PROGRAM P3_03_ProcessData
VAR
	stDBParam 					:ST_ProcessData;	

	fbDBWrite					:FB_PLCDBWriteEvt(sNetId:=CONST.AMS_NETID, tTimeout:=DEFAULT_ADS_TIMEOUT);
	tableColumns				:ARRAY [0..8] OF STRING(50) := ['Batch', 'DateTime', 'Value1', 'Value2', 'Value3', 'Value4', 'Value5', 'Value6', 'Value7'];
	arrParam					:ARRAY [0..8] OF ST_ExpParameter := [(sParaName := 'Batch', nParaSize := 101, eParaType := E_EXPPARAMETERTYPE.STRING_),
															 (sParaName := 'DateTime', nParaSize := 4, eParaType := E_EXPPARAMETERTYPE.DateTime), 
															 (sParaName := 'Value1', nParaSize := 101, eParaType := E_EXPPARAMETERTYPE.STRING_), 
															 (sParaName := 'Value2', nParaSize := 101, eParaType := E_EXPPARAMETERTYPE.STRING_), 
															 (sParaName := 'Value3', nParaSize := 101, eParaType := E_EXPPARAMETERTYPE.STRING_),
															 (sParaName := 'Value4', nParaSize := 101, eParaType := E_EXPPARAMETERTYPE.STRING_),
															 (sParaName := 'Value5', nParaSize := 101, eParaType := E_EXPPARAMETERTYPE.STRING_),
															 (sParaName := 'Value6', nParaSize := 101, eParaType := E_EXPPARAMETERTYPE.STRING_),
															 (sParaName := 'Value7', nParaSize := 101, eParaType := E_EXPPARAMETERTYPE.STRING_)];
		
	fbDeleteTable    			:FB_PLCDBCmdEvt(sNetID:=CONST.AMS_NETID, tTimeout:=DEFAULT_ADS_TIMEOUT);	
	sDelete						:STRING;	
	bDelete						:BOOL;
										 
	bWrite						:BOOL;	
	
	sChopper1Speed				:STRING;
	sChopper2Speed				:STRING;
END_VAR
VAR // added by the converter: edge detectors and wires of the graphical bodies
    _rt1, _rt2 : R_TRIG;
END_VAR

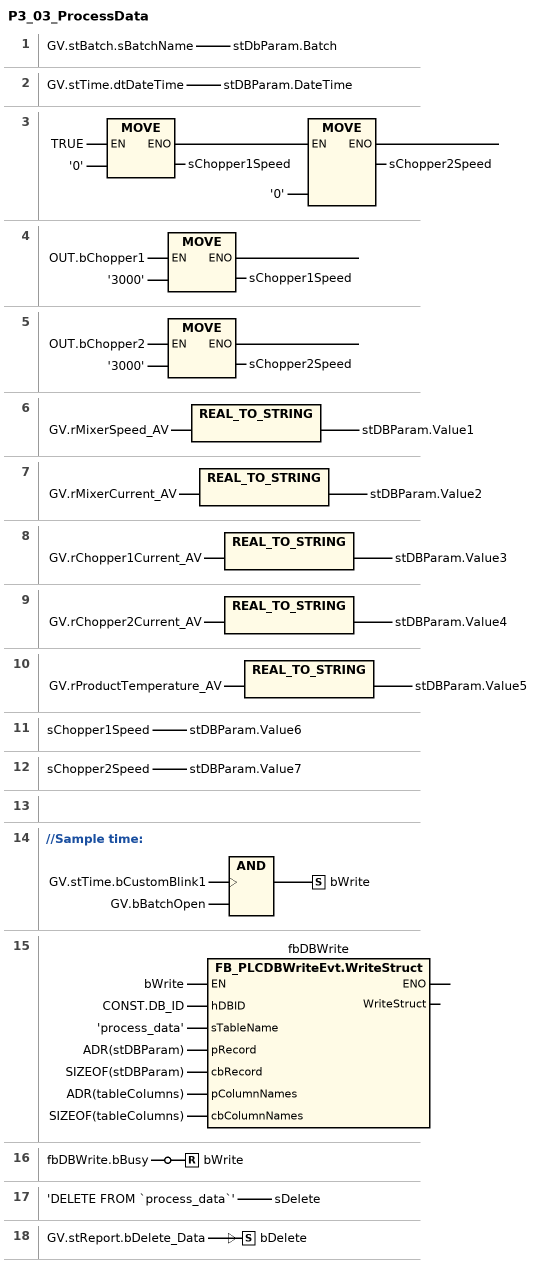
// NETWORK 1
stDbParam.Batch := GV.stBatch.sBatchName;

// NETWORK 2
stDBParam.DateTime := GV.stTime.dtDateTime;

// NETWORK 3
sChopper1Speed := '0';
sChopper2Speed := '0';

// NETWORK 4
IF OUT.bChopper1 THEN sChopper1Speed := '3000'; END_IF

// NETWORK 5
IF OUT.bChopper2 THEN sChopper2Speed := '3000'; END_IF

// NETWORK 6
stDBParam.Value1 := REAL_TO_STRING(GV.rMixerSpeed_AV);

// NETWORK 7
stDBParam.Value2 := REAL_TO_STRING(GV.rMixerCurrent_AV);

// NETWORK 8
stDBParam.Value3 := REAL_TO_STRING(GV.rChopper1Current_AV);

// NETWORK 9
stDBParam.Value4 := REAL_TO_STRING(GV.rChopper2Current_AV);

// NETWORK 10
stDBParam.Value5 := REAL_TO_STRING(GV.rProductTemperature_AV);

// NETWORK 11
stDBParam.Value6 := sChopper1Speed;

// NETWORK 12
stDBParam.Value7 := sChopper2Speed;

// NETWORK 13

// NETWORK 14
// label: //Sample time
_rt1(CLK := GV.stTime.bCustomBlink1);
bWrite S= _rt1.Q AND GV.bBatchOpen;

// NETWORK 15
IF bWrite THEN
    fbDBWrite.WriteStruct(
        hDBID := CONST.DB_ID,
        sTableName := 'process_data',
        pRecord := ADR(stDBParam),
        cbRecord := SIZEOF(stDBParam),
        pColumnNames := ADR(tableColumns),
        cbColumnNames := SIZEOF(tableColumns));
END_IF

// NETWORK 16
bWrite R= NOT fbDBWrite.bBusy;

// NETWORK 17
sDelete := 'DELETE FROM `process_data`';

// NETWORK 18
_rt2(CLK := GV.stReport.bDelete_Data);
bDelete S= _rt2.Q;

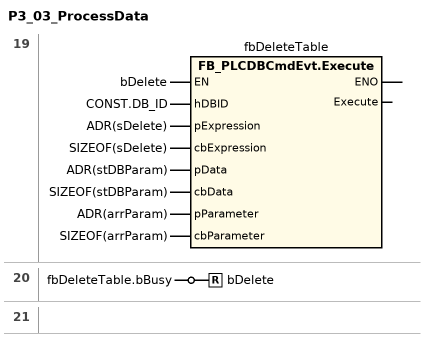
// NETWORK 19
IF bDelete THEN
    fbDeleteTable.Execute(
        hDBID := CONST.DB_ID,
        pExpression := ADR(sDelete),
        cbExpression := SIZEOF(sDelete),
        pData := ADR(stDBParam),
        cbData := SIZEOF(stDBParam),
        pParameter := ADR(arrParam),
        cbParameter := SIZEOF(arrParam));
END_IF

// NETWORK 20
bDelete R= NOT fbDeleteTable.bBusy;

// NETWORK 21

END_PROGRAM

(* stored: Version 1.1.0.1
   POU P3_03_ProcessData: Id {4ea024c6-218b-490f-a3e5-dbb784c2f5cd}, SpecialFunc None *)
